% RSLogix 500 project I2P JOB 16 - SOLUTION.RSS, saved by version 10.00.00.00 %
PROJECT "MWL"    % processor: Bul.1763 MicroLogix 1100 Series B %

PROGRAM FILES
  LAD 2 "MAIN"  7 rungs
  LAD 3 "SIM"  5 rungs  % Simulation %

DATA FILES
  O0 OUTPUT  4 elements
  I1 INPUT  6 elements
  S2 STATUS  66 elements
  B3 BINARY  1 elements
  T4 TIMER  11 elements
  C5 COUNTER  1 elements
  R6 CONTROL  1 elements
  N7 INTEGER  1 elements
  F8 FLOAT  1 elements

LADDER 2 "MAIN"
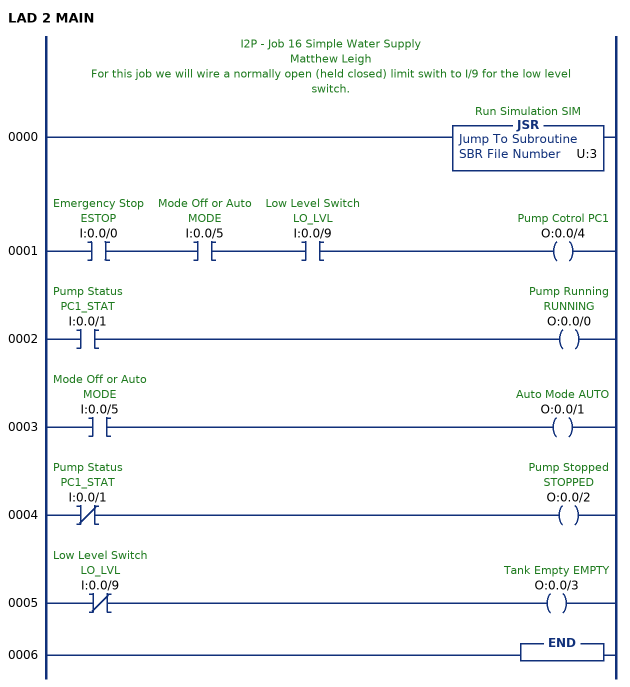
% Rung: 0 %
% I2P - Job 16 Simple Water Supply
% Matthew Leigh
% 
% For this job we will wire a normally open (held closed) limit swith to I/9 for the low level switch. %
SOR JSR U:3 EOR
%   U:3  SIM  "Run Simulation" %
% Rung: 1 %
SOR XIC I:0.0/0 XIC I:0.0/5 XIC I:0.0/9 OTE O:0.0/4 EOR
%   I:0.0/0  ESTOP  "Emergency Stop" %
%   I:0.0/5  MODE  "Mode Off or Auto" %
%   I:0.0/9  LO_LVL  "Low Level Switch" %
%   O:0.0/4  PC1  "Pump Cotrol" %
% Rung: 2 %
SOR XIC I:0.0/1 OTE O:0.0/0 EOR
%   I:0.0/1  PC1_STAT  "Pump Status" %
%   O:0.0/0  RUNNING  "Pump Running" %
% Rung: 3 %
SOR XIC I:0.0/5 OTE O:0.0/1 EOR
%   I:0.0/5  MODE  "Mode Off or Auto" %
%   O:0.0/1  AUTO  "Auto Mode" %
% Rung: 4 %
SOR XIO I:0.0/1 OTE O:0.0/2 EOR
%   I:0.0/1  PC1_STAT  "Pump Status" %
%   O:0.0/2  STOPPED  "Pump Stopped" %
% Rung: 5 %
SOR XIO I:0.0/9 OTE O:0.0/3 EOR
%   I:0.0/9  LO_LVL  "Low Level Switch" %
%   O:0.0/3  EMPTY  "Tank Empty" %
% Rung: 6 %
SOR END EOR

LADDER 3 "SIM"    % Simulation %
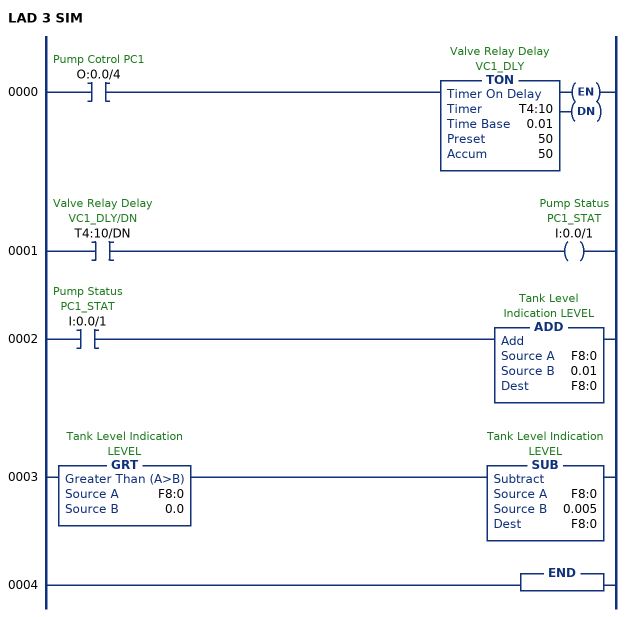
% Rung: 0 %
SOR XIC O:0.0/4 TON T4:10 0.01 50 50 EOR
%   O:0.0/4  PC1  "Pump Cotrol" %
%   T4:10  VC1_DLY  "Valve Relay Delay" %
% Rung: 1 %
SOR XIC T4:10/DN OTE I:0.0/1 EOR
%   T4:10  VC1_DLY  "Valve Relay Delay" %
%   I:0.0/1  PC1_STAT  "Pump Status" %
% Rung: 2 %
SOR XIC I:0.0/1 ADD F8:0 0.01 F8:0 EOR
%   I:0.0/1  PC1_STAT  "Pump Status" %
%   F8:0  LEVEL  "Tank Level Indication" %
% Rung: 3 %
SOR GRT F8:0 0.0 SUB F8:0 0.005 F8:0 EOR
%   F8:0  LEVEL  "Tank Level Indication" %
% Rung: 4 %
SOR END EOR

DATA TABLE (non-zero values as saved)
DATA T4
% .PRE .ACC %
% T4:10 % 50 50
DATA F8
% F8:0 % 13.94172
